// Encodes and writes a tag.
FUNCTION F_WriteTag : HRESULT
VAR_IN_OUT      
    stCtx : ST_WriteContext;
END_VAR
VAR_INPUT
    nFieldNumber    : UDINT;
    eWireType       : E_WireType;
END_VAR
VAR 
    nTag : UDINT;
END_VAR

nTag := F_MakeTag(nFieldNumber, eWireType);
F_WriteTag := F_WriteRawVarint32(stCtx, nTag);

END_FUNCTION

(* stored: Version 1.1.0.1
   POU F_WriteTag: Id {ae3ccd4b-1305-434e-9f0c-c1a8e3523e7a}, SpecialFunc None *)
